{attribute 'GeneratedUsingTerminal: ER5101-0002-0019'}
{attribute addProperty BoxType "ER5101-0002-0019"}
{attribute addProperty Id "StatusAT %I*Status_3A9E406C12Counter_valueAT %I*UINT2Latch_valueAT %I*UINT2"}
{attribute addProperty CRC "4109931907"}
{attribute addProperty Size "16"}
TYPE ENC_Status_compact_F4F89583 :
STRUCT
	{attribute addProperty Name "Status"}
	Status AT %I* : Status_3A9E406C;
	{attribute addProperty Name "Counter_value"}
	Counter_value AT %I* : UINT;
	{attribute addProperty Name "Latch_value"}
	Latch_value AT %I* : UINT;
END_STRUCT
END_TYPE

(* stored: Version 1.2.0.0, ProductVersion 3.1.4024.9
   DUT ENC_Status_compact_F4F89583: Id {b1931ab5-9424-4944-8fbd-0246cbfa40f9} *)
